{attribute 'linkalways'} 
{attribute 'no_explicit_call' := 'This FB is a CLASS and must be accessed using methods or properties'}
{attribute 'enable_dynamic_creation'}
FUNCTION_BLOCK Node_F_VN_ContainerAverageVarianceElementwise3 EXTENDS VisionNode
VAR
    ipSrcContainer : _ITcVnContainer;
    aAverage : _TcVnVector3_LREAL;
	aVariance : _TcVnVector3_LREAL;
    hrPrev : _HRESULT(S_OK);
    hresult : _HRESULT(S_OK);
END_VAR

METHOD PUBLIC  Clone : I_Node
VAR
	pNode : POINTER TO Node_F_VN_ContainerAverageVarianceElementwise3;
END_VAR
pNode := __NEW(Node_F_VN_ContainerAverageVarianceElementwise3);
Clone := pNode^;
END_METHOD

METHOD FB_init : BOOL
VAR_INPUT
	bInitRetains : BOOL; // if TRUE, the retain variables are initialized (warm start / cold start)
	bInCopyCode : BOOL;  // if TRUE, the instance afterwards gets moved into the copy code (online change)
END_VAR
AddInput('ipSrcContainer', ipSrcContainer);
AddInput('hrPrev', hrPrev);
AddOutput('aAverage', aAverage);
AddOutput('aVariance', aVariance);
AddOutput('hresult',hresult);
END_METHOD

METHOD PROTECTED OnExecute
hresult.Value := F_VN_ContainerAverageVarianceElementwise3(
    ipSrcContainer := ipSrcContainer.Value,
    aAverage := aAverage.Value,
	aVariance := aVariance.Value,
    hrPrev:= hrPrev.Value);
END_METHOD

METHOD PUBLIC PreExecutionCheck
VAR_INPUT
	Check : I_PreExecutionChecks;
END_VAR
VAR
	isCorrectType : BOOL;
END_VAR
Check.IsTrue(ipSrcContainer.IsValid, 'ipContainer must be a valid container');

isCorrectType := 
    // ---------------------------------------------------------
    // Point 3 Types (X, Y, Z)
    // ---------------------------------------------------------
    ipSrcContainer.IsType(TC_GLOBAL_CONST_LIST.ContainerType_Vector_TcVnPoint3_REAL) OR_ELSE
    ipSrcContainer.IsType(TC_GLOBAL_CONST_LIST.ContainerType_Vector_TcVnPoint3_LREAL) OR_ELSE

    // ---------------------------------------------------------
    // Vector 3 Types (X, Y, Z)
    // ---------------------------------------------------------
    ipSrcContainer.IsType(TC_GLOBAL_CONST_LIST.ContainerType_Vector_TcVnVector3_SINT) OR_ELSE
    ipSrcContainer.IsType(TC_GLOBAL_CONST_LIST.ContainerType_Vector_TcVnVector3_USINT) OR_ELSE
    ipSrcContainer.IsType(TC_GLOBAL_CONST_LIST.ContainerType_Vector_TcVnVector3_INT) OR_ELSE
    ipSrcContainer.IsType(TC_GLOBAL_CONST_LIST.ContainerType_Vector_TcVnVector3_UINT) OR_ELSE
    ipSrcContainer.IsType(TC_GLOBAL_CONST_LIST.ContainerType_Vector_TcVnVector3_REAL);

Check.IsTrue(isCorrectType, 'ipContainer contains incorrect type for Elementwise3');
END_METHOD

END_FUNCTION_BLOCK

(* stored: Version 1.1.0.1, ProductVersion 3.1.4026.13
   POU Node_F_VN_ContainerAverageVarianceElementwise3: Id {ae1fe61d-cdae-019e-17ef-9653c27b1007}, SpecialFunc None
   Folder Constructor: Id {e86241e8-9def-089e-3482-d9214e2017a0}
   Method Clone: Id {c9d726a2-f422-0c9b-11d6-a958553e7438}
   Method FB_init: Id {09ddb2bf-e02a-0ce4-0630-419b211029b7}
   Method OnExecute: Id {443c133d-4d5d-03f1-12be-319bff726799}
   Method PreExecutionCheck: Id {e422de0f-5842-05b1-0e58-9d32704c312e} *)
